% RSLogix 500 project I2P Job 15 - Tyler_Vogt.RSS, saved by version 10.00.00.00 %
PROJECT "MLO2B"    % processor: Bul.1763 MicroLogix 1100 Series B %

PROGRAM FILES
  LAD 2   15 rungs

DATA FILES
  O0 OUTPUT  4 elements
  I1 INPUT  6 elements
  S2 STATUS  66 elements
  B3 BINARY  1 elements
  T4 TIMER  2 elements
  C5 COUNTER  1 elements
  R6 CONTROL  1 elements
  N7 INTEGER  1 elements
  F8 FLOAT  1 elements

LADDER 2
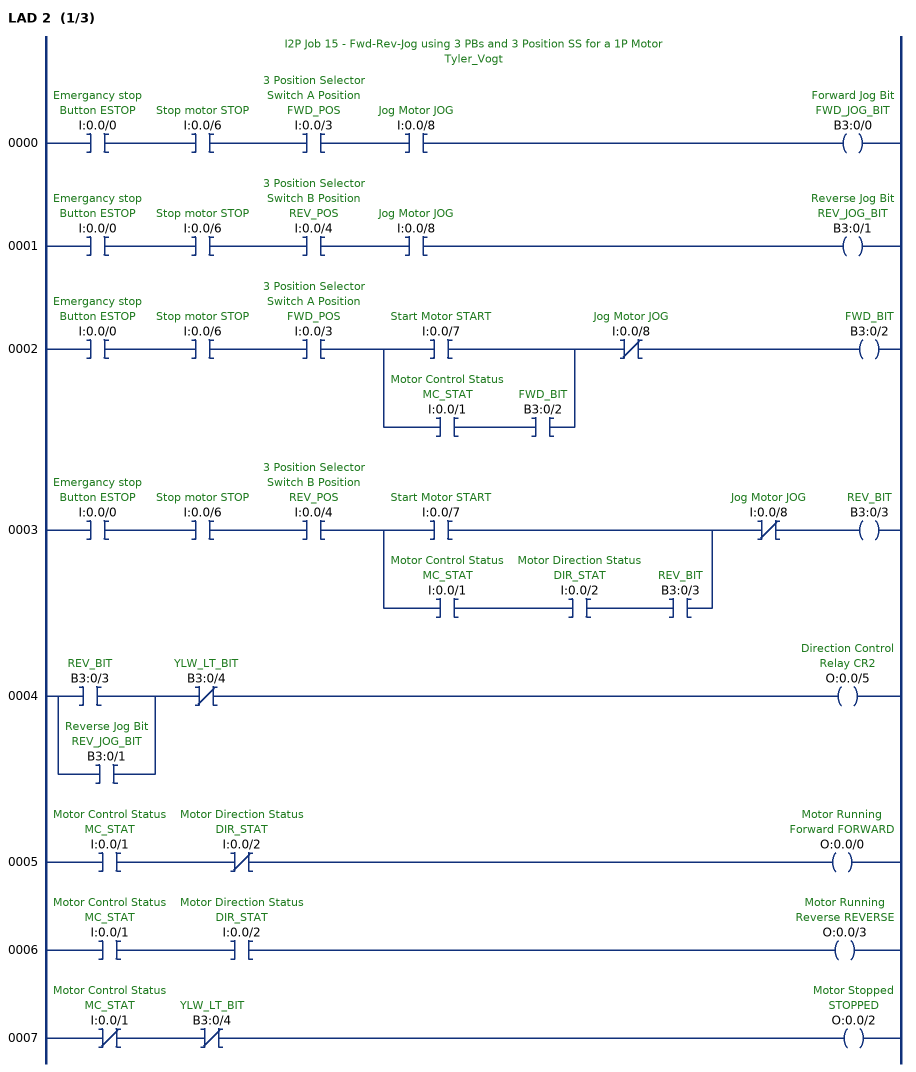
% Rung: 0 %
% I2P Job 15 - Fwd-Rev-Jog using 3 PBs and 3 Position SS for a 1P Motor
% Tyler_Vogt %
SOR XIC I:0.0/0 XIC I:0.0/6 XIC I:0.0/3 XIC I:0.0/8 OTE B3:0/0 EOR
%   I:0.0/0  ESTOP  "Emergancy stop Button" %
%   I:0.0/6  STOP  "Stop motor" %
%   I:0.0/3  FWD_POS  "3 Position Selector Switch A Position" %
%   I:0.0/8  JOG  "Jog Motor" %
%   B3:0/0  FWD_JOG_BIT  "Forward Jog Bit" %
% Rung: 1 %
SOR XIC I:0.0/0 XIC I:0.0/6 XIC I:0.0/4 XIC I:0.0/8 OTE B3:0/1 EOR
%   I:0.0/0  ESTOP  "Emergancy stop Button" %
%   I:0.0/6  STOP  "Stop motor" %
%   I:0.0/4  REV_POS  "3 Position Selector Switch B Position" %
%   I:0.0/8  JOG  "Jog Motor" %
%   B3:0/1  REV_JOG_BIT  "Reverse Jog Bit" %
% Rung: 2 %
SOR XIC I:0.0/0 XIC I:0.0/6 XIC I:0.0/3 BST XIC I:0.0/7 NXB XIC I:0.0/1 XIC B3:0/2 BND XIO I:0.0/8 OTE B3:0/2 EOR
%   I:0.0/0  ESTOP  "Emergancy stop Button" %
%   I:0.0/6  STOP  "Stop motor" %
%   I:0.0/3  FWD_POS  "3 Position Selector Switch A Position" %
%   I:0.0/7  START  "Start Motor" %
%   I:0.0/1  MC_STAT  "Motor Control Status" %
%   B3:0/2  FWD_BIT %
%   I:0.0/8  JOG  "Jog Motor" %
% Rung: 3 %
SOR XIC I:0.0/0 XIC I:0.0/6 XIC I:0.0/4 BST XIC I:0.0/7 NXB XIC I:0.0/1 XIC I:0.0/2 XIC B3:0/3 BND XIO I:0.0/8 OTE B3:0/3 EOR
%   I:0.0/0  ESTOP  "Emergancy stop Button" %
%   I:0.0/6  STOP  "Stop motor" %
%   I:0.0/4  REV_POS  "3 Position Selector Switch B Position" %
%   I:0.0/7  START  "Start Motor" %
%   I:0.0/1  MC_STAT  "Motor Control Status" %
%   I:0.0/2  DIR_STAT  "Motor Direction Status" %
%   B3:0/3  REV_BIT %
%   I:0.0/8  JOG  "Jog Motor" %
% Rung: 4 %
SOR BST XIC B3:0/3 NXB XIC B3:0/1 BND XIO B3:0/4 OTE O:0.0/5 EOR
%   B3:0/3  REV_BIT %
%   B3:0/1  REV_JOG_BIT  "Reverse Jog Bit" %
%   B3:0/4  YLW_LT_BIT %
%   O:0.0/5  CR2  "Direction Control Relay" %
% Rung: 5 %
SOR XIC I:0.0/1 XIO I:0.0/2 OTE O:0.0/0 EOR
%   I:0.0/1  MC_STAT  "Motor Control Status" %
%   I:0.0/2  DIR_STAT  "Motor Direction Status" %
%   O:0.0/0  FORWARD  "Motor Running Forward" %
% Rung: 6 %
SOR XIC I:0.0/1 XIC I:0.0/2 OTE O:0.0/3 EOR
%   I:0.0/1  MC_STAT  "Motor Control Status" %
%   I:0.0/2  DIR_STAT  "Motor Direction Status" %
%   O:0.0/3  REVERSE  "Motor Running Reverse" %
% Rung: 7 %
SOR XIO I:0.0/1 XIO B3:0/4 OTE O:0.0/2 EOR
%   I:0.0/1  MC_STAT  "Motor Control Status" %
%   B3:0/4  YLW_LT_BIT %
%   O:0.0/2  STOPPED  "Motor Stopped" %

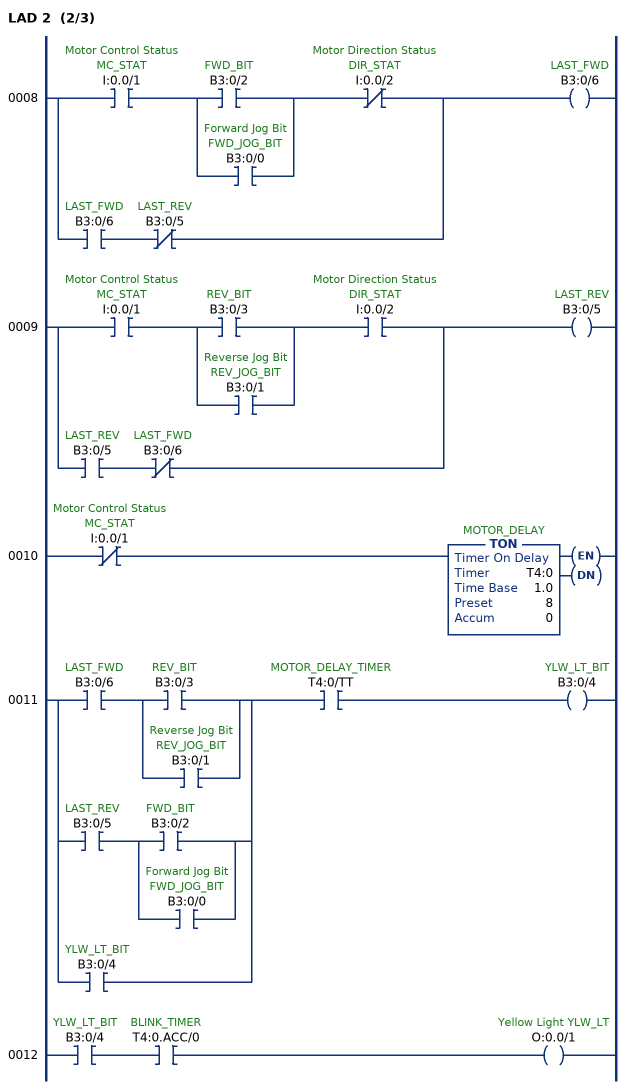
% Rung: 8 %
SOR BST XIC I:0.0/1 BST XIC B3:0/2 NXB XIC B3:0/0 BND XIO I:0.0/2 NXB XIC B3:0/6 XIO B3:0/5 BND OTE B3:0/6 EOR
%   I:0.0/1  MC_STAT  "Motor Control Status" %
%   B3:0/2  FWD_BIT %
%   B3:0/0  FWD_JOG_BIT  "Forward Jog Bit" %
%   I:0.0/2  DIR_STAT  "Motor Direction Status" %
%   B3:0/6  LAST_FWD %
%   B3:0/5  LAST_REV %
% Rung: 9 %
SOR BST XIC I:0.0/1 BST XIC B3:0/3 NXB XIC B3:0/1 BND XIC I:0.0/2 NXB XIC B3:0/5 XIO B3:0/6 BND OTE B3:0/5 EOR
%   I:0.0/1  MC_STAT  "Motor Control Status" %
%   B3:0/3  REV_BIT %
%   B3:0/1  REV_JOG_BIT  "Reverse Jog Bit" %
%   I:0.0/2  DIR_STAT  "Motor Direction Status" %
%   B3:0/5  LAST_REV %
%   B3:0/6  LAST_FWD %
% Rung: 10 %
SOR XIO I:0.0/1 TON T4:0 1.0 8 0 EOR
%   I:0.0/1  MC_STAT  "Motor Control Status" %
%   T4:0  MOTOR_DELAY %
% Rung: 11 %
SOR BST BST XIC B3:0/6 BST XIC B3:0/3 NXB XIC B3:0/1 BND NXB XIC B3:0/5 BST XIC B3:0/2 NXB XIC B3:0/0 BND BND NXB XIC B3:0/4 BND XIC T4:0/TT OTE B3:0/4 EOR
%   B3:0/6  LAST_FWD %
%   B3:0/3  REV_BIT %
%   B3:0/1  REV_JOG_BIT  "Reverse Jog Bit" %
%   B3:0/5  LAST_REV %
%   B3:0/2  FWD_BIT %
%   B3:0/0  FWD_JOG_BIT  "Forward Jog Bit" %
%   B3:0/4  YLW_LT_BIT %
%   T4:0/TT  MOTOR_DELAY_TIMER %
% Rung: 12 %
SOR XIC B3:0/4 XIC T4:0.ACC/0 OTE O:0.0/1 EOR
%   B3:0/4  YLW_LT_BIT %
%   T4:0.ACC/0  BLINK_TIMER %
%   O:0.0/1  YLW_LT  "Yellow Light" %

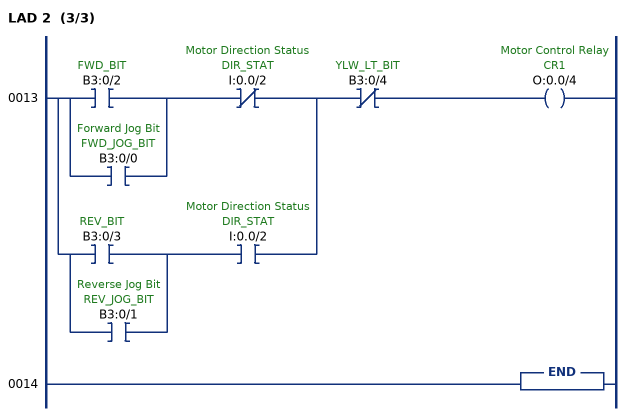
% Rung: 13 %
SOR BST BST XIC B3:0/2 NXB XIC B3:0/0 BND XIO I:0.0/2 NXB BST XIC B3:0/3 NXB XIC B3:0/1 BND XIC I:0.0/2 BND XIO B3:0/4 OTE O:0.0/4 EOR
%   B3:0/2  FWD_BIT %
%   B3:0/0  FWD_JOG_BIT  "Forward Jog Bit" %
%   I:0.0/2  DIR_STAT  "Motor Direction Status" %
%   B3:0/3  REV_BIT %
%   B3:0/1  REV_JOG_BIT  "Reverse Jog Bit" %
%   B3:0/4  YLW_LT_BIT %
%   O:0.0/4  CR1  "Motor Control Relay" %
% Rung: 14 %
SOR END EOR

OTHER DOCUMENTED ADDRESSES
  B3:0/7  STOP_BIT  "Estop and Stop"
  FWD_JOG  "Forward Jog"
  I:0.0/5  RUN_JOG  "2 Position Selector Switch A Position"
  MOTOR  
  T4:1  FWD_DELAY

DATA TABLE (non-zero values as saved)
DATA B3
% B3:0 % 0X0004
DATA T4
% .PRE .ACC %
% T4:0 % 8 0
% T4:1 % 8 0
